{attribute 'qualified_only'}
VAR_GLOBAL PERSISTENT
	fJointPositionOffset 	: ARRAY [0..2] OF LREAL;	
	fJointCalibrationOffset : ARRAY [0..2] OF LREAL;
END_VAR

(* stored: Version 1.1.0.1, ProductVersion 3.1.4024.3
   GVL Parameters: Id {11109a4f-d22d-4ff0-beff-18bcb47d8d61} *)
